(* PLC project 117_1_V0.5.project, CODESYS CODESYS V3.5 SP17 Patch 3 *)
(* stored: creationDateTime 1970-01-01T00:00:00, modificationDateTime 2026-06-16T22:51:19.9979415 *)

FUNCTION_BLOCK BasicPIDController
  VAR
    _Pv : REAL;
    _Sp : REAL;
    _Kp : REAL;
    _Ki : REAL;
    _Kd : REAL;
    _Ts : TIME;
    _Error : REAL;
    _Output : REAL;
    _MinOut : REAL;
    _MaxOut : REAL;
    _Direction : PID_DIRECTION_UDT;
    _PreviousError : REAL;
    _Proportional : REAL;
    _Integral : REAL;
    _Differential : REAL;
    _Status : PID_STATUS_UDT;
  END_VAR

            //Включение ПИД
IF _Status <> Enabled THEN
	Reset();	//Integral := 0; PreviousError := 0;Output := 0;
	RETURN;
ELSE
//Значение текущей ошибки
_Error			:= xError(); //CASE Direction OF DIRECT:xError := (Sp - Pv) * 1.0; REVERSE:xError := (Sp - Pv) * -1.0; END_CASE
// Пропорционал
_Proportional	:= xProportional();	//xProportional := Kp * Error;
// Интеграл
_Integral		:= xIntegral();	//xIntegral := LIMIT(OutMin, (Integral + Ki * Error * ((TIME_TO_REAL (Ts)) / 1000)), OutMax);
// ДиФФеренциал
_Differential	:= xDifferential(); //xDifferential := Kd * (Error - PreviousError) / ((TIME_TO_REAL (Ts)) / 1000);
//Значение предыдущей ошибки
_PreviousError	:= _Error;
//Выход ПИД
_Output := LIMIT(_MinOut, _Proportional + _Integral + _Differential, _MaxOut);
END_IF




          

METHOD Set_Configuration : BOOL
  VAR_INPUT
    Kp : REAL := 0.1;
    Ki : REAL := 0;
    Kd : REAL := 0;
    Ts : TIME := TIME#100ms;
    MinOut : REAL := 0;
    MaxOut : REAL := 100;
    Direction : PID_DIRECTION_UDT := DIRECT;
  END_VAR
                  _Kp 		 := Kp;		
_Ki 		 := Ki;		
_Kd 		 := Kd;		
_Ts			 := Ts;		
_MinOut		 := MinOut;		
_MaxOut		 := MaxOut;	
_Direction   := Direction;
                
END_METHOD

METHOD Get_Diagnostics : PID_DIAGNOSTIC_UDT
                  Get_Diagnostics.Error			:= _Error;			      
Get_Diagnostics.PreviousError	:= _PreviousError;			
Get_Diagnostics.Proportional	:= _Proportional;	 		
Get_Diagnostics.Integral		:= _Integral;		    	
Get_Diagnostics.Differential	:= _Differential;	 		
Get_Diagnostics.Direction		:= _Direction;		   	
Get_Diagnostics.Status			:= _Status;			     
Get_Diagnostics.Kp 				:= _Kp; 		  
Get_Diagnostics.Ki 				:= _Ki; 		  
Get_Diagnostics.Kd 				:= _Kd; 		  
Get_Diagnostics.Ts				:= _Ts;	   
Get_Diagnostics.MinOut			:= _MinOut;	
Get_Diagnostics.MaxOut			:= _MaxOut;	
    
                
END_METHOD

METHOD xDifferential : REAL
                  xDifferential := _Kd * (_Error - _PreviousError) / ((TIME_TO_REAL (_Ts)) / 1000);
                
END_METHOD

METHOD Enable : BOOL
                  _Status := Enabled;

                
END_METHOD

METHOD Disable : BOOL
                  _Status := Disabled;
                
END_METHOD

METHOD xError : REAL
                  CASE _Direction OF
DIRECT:
	xError := (_Sp - _Pv) * 1.0;
REVERSE:
	xError := (_Sp - _Pv) * -1.0;
END_CASE
                
END_METHOD

METHOD xIntegral : REAL
                  xIntegral := LIMIT(_MinOut, (_Integral + _Ki * _Error * ((TIME_TO_REAL (_Ts)) / 1000)), _MaxOut);
                
END_METHOD

METHOD Reset : BOOL
                  _Error			:= 0;
_Integral		:= 0;
_PreviousError	:= 0;
_Output 		:= 0;
                
END_METHOD

METHOD xProportional : REAL
                  xProportional := _Kp * _Error;
                
END_METHOD

PROPERTY xSp : REAL
GET
                    xSp := _Sp;
                  
END_GET
SET
                    _Sp := xSp;
                  
END_SET
END_PROPERTY

PROPERTY xPv : REAL
GET
                    xPv := _Pv;
                  
END_GET
SET
                    _Pv := xPv;
                  
END_SET
END_PROPERTY

PROPERTY xOutput : REAL
GET
                    xOutput := _Output;
                  
END_GET
SET
                    
                  
END_SET
END_PROPERTY
END_FUNCTION_BLOCK
